TYPE SAFETY_IN :
STRUCT

	DOORS_FBerr:BOOL;
	DOORS_COMerr:BOOL;
	DOORS_State:USINT;
	DOOR_VAC_CLOSED:BOOL;
	DOOR_Q1_CLOSED:BOOL;
	DOOR_Q2_CLOSED:BOOL;
	DOOR_PMAX_CLOSED:BOOL;
	DOOR_PRINT_CLOSED:BOOL;

	NOT_AUS_FBerr:BOOL;
	NOT_AUS_COMerr:BOOL;
	NOT_AUS_State:USINT;

END_STRUCT
END_TYPE

(* stored: Version 1.1.0.1, ProductVersion 3.1.0.26
   DUT SAFETY_IN: Id {97f806cc-bc7a-4a21-8900-b13c8c95a3e3} *)
